FUNCTION_BLOCK RegulationParametersFB
VAR_IN_OUT
	Parameters: GreenMasterBaseParameters;
END_VAR
VAR_INPUT
	Control: RegulationControlParameters;
	SupplyAir: AirParametersFB := (StartupFanSpeed := 0.3, SetPointAdjustment := (Curve := (Y1 := 165, Y2 := 165, Y3 := 165, Y4 := 165, Y5 := 165, Y6 := 165, Y7 := 165, Y8 := 165, Y9 := 165)));
	ExtractAir: AirParametersFB := (StartupFanSpeed := 0.4, SetPointAdjustment := (Curve := (Y1 := 160, Y2 := 160, Y3 := 160, Y4 := 160, Y5 := 160, Y6 := 160, Y7 := 160, Y8 := 160, Y9 := 160)));
	Temperature: TemperatureControlParametersFB;
	NightCoolingLimit: LREAL;
	TemperatureCompensationSource: TemperatureCompensationSources;
	CurrentTemperatureCompensationSource: TemperatureCompensationSources;
	CompensationTemperature: LREAL;
	SystemSpecificFanPower: LREAL; // $(unit "kPa")
	SystemEfficiency: LREAL; // $(scale "0 1 0 100", unit "%")
END_VAR
VAR_OUTPUT
END_VAR
VAR
	CurrentMaxFlow: LREAL;
END_VAR

SupplyAir(Parameters := Parameters);
ExtractAir(Parameters := Parameters);
Temperature(Parameters := Parameters, EN:=Parameters.System.Operation.EN);

IF __ISVALIDREF(Parameters.GetGreenMaster()) THEN
	Temperature.Control.PV := Parameters.GetGreenMaster().GetCurrentPV();
	SupplyAir.Control.PV := Parameters.GetGreenMaster().GetCurrentSupplyAirPV();
	ExtractAir.Control.PV := Parameters.GetGreenMaster().GetCurrentExtractAirPV();
END_IF

CASE TemperatureCompensationSource OF
	TemperatureCompensationSources.Auto:
		CompensationTemperature := Parameters.IO.AIn.BT1;
		IF (NOT Parameters.IO.AIn.BT1_EN) OR Parameters.IO.AIn.BT1_Error THEN
			CompensationTemperature := Parameters.IO.AIn.T_BT2;
			CurrentTemperatureCompensationSource := TemperatureCompensationSources.T_BT2;
		ELSE
			CurrentTemperatureCompensationSource := TemperatureCompensationSources.BT1;			
		END_IF;
	TemperatureCompensationSources.BT1:
		CurrentTemperatureCompensationSource := TemperatureCompensationSources.BT1;
		CompensationTemperature := Parameters.IO.AIn.BT1;
	TemperatureCompensationSources.T_BT2:
		CurrentTemperatureCompensationSource := TemperatureCompensationSources.T_BT2;
		CompensationTemperature := Parameters.IO.AIn.T_BT2;
END_CASE
SupplyAir.Flow := Parameters.IO.AIn.T_BF1;
ExtractAir.Flow := Parameters.IO.AIn.F_BF1;
SupplyAir.Power := Main.GreenMaster.AI2.T_CurrentPower;
ExtractAir.Power := Main.GreenMaster.AI2.F_CurrentPower;
SupplyAir.PressureRise := Parameters.IO.AIn.T_BF1;
ExtractAir.PressureRise := Parameters.IO.AIn.F_BF1;
CurrentMaxFlow := MAX(ExtractAir.Flow, SupplyAir.Flow);
IF CurrentMaxFlow <> 0 THEN
	SystemSpecificFanPower := (ExtractAir.Power + SupplyAir.Power) / CurrentMaxFlow;	
ELSE
	SystemSpecificFanPower := 0;
END_IF
IF (SupplyAir.PressureRise + ExtractAir.PressureRise) <> 0 THEN
	SystemEfficiency := (SupplyAir.SpecificFanPower + ExtractAir.SpecificFanPower) / ((SupplyAir.PressureRise + ExtractAir.PressureRise) / 1000);
ELSE
	SystemEfficiency := 0;	
END_IF

END_FUNCTION_BLOCK

(* stored: Version 1.1.0.1, ProductVersion 3.1.4024.6
   POU RegulationParametersFB: Id {35458062-23b8-41fa-a7d8-32b0bd66ddbe}, SpecialFunc None *)
